Yaskawa INFORM job: ERROR.JBI

/JOB
//NAME ERROR
//POS
///NPOS 0,0,0,0,0,0
//INST
///DATE 2018/11/14 12:52
///ATTR SC,RW,SY
///LVARS 1,0,0,0,0,0,0,0
NOP
*TOP
'*****
DIN LB000 SOUT#(5)
IFTHEN LB000=1
	 DOUT OG#(74) 4
ENDIF
'*****
IFTHEN B003=1
	 DOUT OG#(74) 1
ENDIF
'*****
IFTHEN B003=5
	 DOUT OG#(74) 5
ENDIF
'*****
IFTHEN B003=8
	 DOUT OG#(74) 8
ENDIF
'*****
IFTHEN LB000=0 ANDIF B003=0
	 DOUT OG#(74) 0
ENDIF
DELAY 20
JUMP *TOP
END
